{attribute 'GeneratedUsingTerminal: EP2816-0004-0016'}
{attribute addProperty BoxType "EP2816-0004-0016"}
{attribute addProperty Id "DO_Outputs_Channel_1AT %Q*DO_Outputs_Channel_28AC1A9E8DO_Outputs_Channel_2AT %Q*DO_Outputs_Channel_28AC1A9E8WcStateAT %I*WcState_0B2B16F91InfoDataAT %I*InfoData_94A18F5E2"}
{attribute addProperty CRC "1726561023"}
{attribute addProperty Size "19"}
TYPE EP2816_66E93AFF EXTENDS EtcSlaveTerminalBase_947E5A46 :
STRUCT
	{attribute addProperty Name "DO_Outputs_Channel_1"}
	DO_Outputs_Channel_1 : DO_Outputs_Channel_28AC1A9E;
	{attribute addProperty Name "DO_Outputs_Channel_2"}
	DO_Outputs_Channel_2 : DO_Outputs_Channel_28AC1A9E;
	{attribute addProperty Name "WcState"}
	WcState : WcState_0B2B16F9;
	{attribute addProperty Name "InfoData"}
	InfoData : InfoData_94A18F5E;
END_STRUCT
END_TYPE

(* stored: Version 1.2.0.0, ProductVersion 3.1.4024.9
   DUT EP2816_66E93AFF: Id {b5e83a23-51a0-440b-bab9-f9b2ff6e35d7} *)
